TYPE AX5000_P_1000 :
STRUCT
	Debug_pointer_1_adr:UDINT;
END_STRUCT
END_TYPE

(* stored: Version 1.1.0.1, ProductVersion 3.1.4024.3
   DUT AX5000_P_1000: Id {b11eb4c4-5c50-44b4-b3f9-b82bd6538a96} *)
